TYPE TcoTixonPickVibroBasic_Control_v_1_x_x EXTENDS TcoTixonGenericControl : STRUCT
END_STRUCT
END_TYPE

(* stored: Version 1.1.0.1, ProductVersion 3.1.4024.12
   DUT TcoTixonPickVibroBasic_Control_v_1_x_x: Id {bf9e881a-eb59-07c2-0fd4-331dba64a02b} *)
